# EPICS autosave request: iocBoot/sioc-b084-bl04/blen_manual.req
file "lcls2_gap_manual.req" AREA=HTR,POS=350,INST=0
file "lcls2_gap_manual.req" AREA=HTR,POS=350,INST=1
